Staubli VAL3: start.pgx

program start()
begin

  call init()
  taskCreate "PLC",100,cycle:_tPLC()
  taskCreate "HIM",100,libload("Disk://page/page_viewTraj")
  taskCreate "_WatchDog",100,cycle:_WatchDog()
  // call WatchDog()

end
